Omron CX-Programmer project 新工程 (CX-Programmer 9.73)

# PLC 新PLC1: CPM2* 

## Global symbols (name address type ; comment)
0.00 BOOL  ; 系统工作/停止开
0.01 BOOL  ; 温度过高报警信号
0.03 BOOL  ; 湿度过高报警信号
0.05 BOOL  ; 烟雾报警信号
10.00 BOOL  ; 1
10.01 BOOL  ; 排风扇
10.02 BOOL  ; 烟雾报警信号
10.03 BOOL  ; 温度报警信号
10.04 BOOL  ; 系统运行灯
10.05 BOOL  ; 温度报警灯
10.06 BOOL  ; 湿度报警灯
10.07 BOOL  ; 烟雾报警灯
200.00 BOOL  ; 0点开信号
200.01 BOOL  ; 4点开信号
200.02 BOOL  ; 8点开信号
200.03 BOOL  ; 12点开信号
200.04 BOOL  ; 16点开信号
200.05 BOOL  ; 20点开信号
200.10 BOOL  ; 触发信号
232.00 BOOL  ; 系统运行

## Program 新程序1 (no task)
; 原创、欧姆龙PLC、CPM2A自身时钟六个时间段触发程序 / 简单程序，高手请飘过。 / 欧姆龙CPM2A六个时间段触发程序。 / 触发时间为0点，4点，8点，12点，16点，20点（可通过修改CMP20#的值修改触发时间）一分钟后断开。 / 触发次数也可通过增减CMP20来实现。 / 在实际应用中，当系统工作开关开启时，系统根据PLC时钟读取时间数据，在 0点、4点、8点、12点、16点、20点 置位对应的触发信号，并通过这些信号组合生成综合触发信号来驱动设备动作。当综合触发信号被置位时，系统进入运行状态并准备设备动作。系统确保在任一时刻，只有一个触发信号被置位，以保证动作独立执行。 / 系统还集成了安全监测功能，当温度过高信号、湿度过高信号或烟雾检测信号被触发时，温度报警灯、湿度报警灯或烟雾报警灯会点亮，同时通过温度报警输出或烟雾报警输出通知外部设备，以保护生产安全。若 0点触发信号被置位，启动设备初始动作；若 4点触发信号被置位，调整设备运行参数。此外，PLC时钟与实际时间保持同步，在 0点 准时置位 0点触发信号，准备设备运行。

### Section 段1

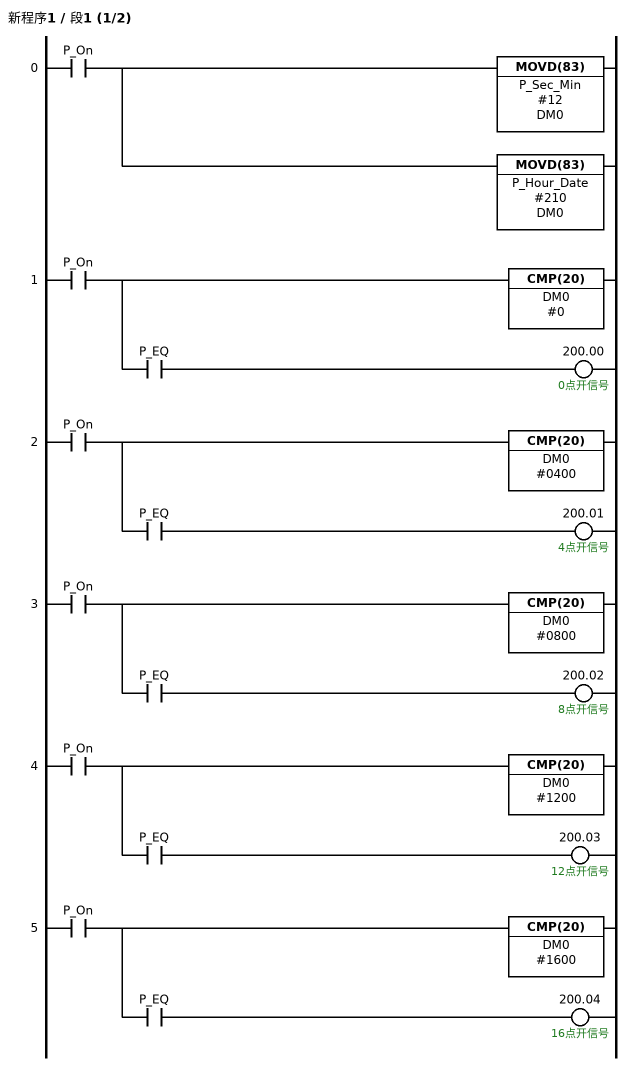
; rung 0
LD P_On
MOVD(83) P_Sec_Min #12 DM0
MOVD(83) P_Hour_Date #210 DM0
; rung 1
LD P_On
CMP(20) DM0 #0
AND P_EQ
OUT 200.00  ; 0点开信号
; rung 2
LD P_On
CMP(20) DM0 #0400
AND P_EQ
OUT 200.01  ; 4点开信号
; rung 3
LD P_On
CMP(20) DM0 #0800
AND P_EQ
OUT 200.02  ; 8点开信号
; rung 4
LD P_On
CMP(20) DM0 #1200
AND P_EQ
OUT 200.03  ; 12点开信号
; rung 5
LD P_On
CMP(20) DM0 #1600
AND P_EQ
OUT 200.04  ; 16点开信号

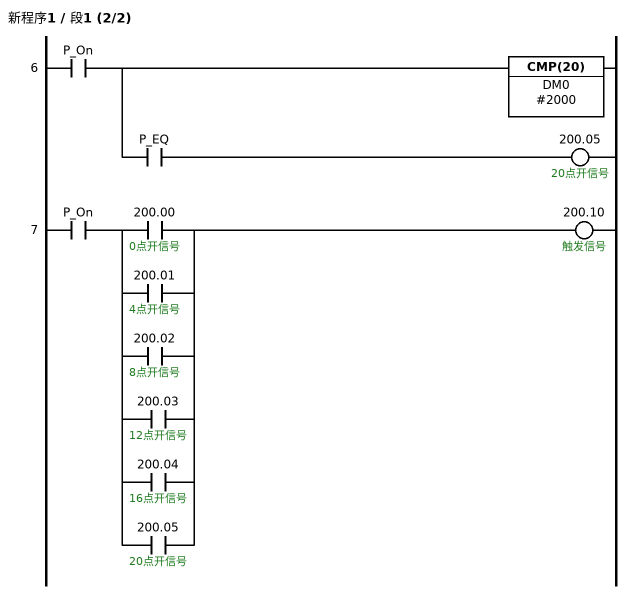
; rung 6
LD P_On
CMP(20) DM0 #2000
AND P_EQ
OUT 200.05  ; 20点开信号
; rung 7
LD P_On
LD 200.00  ; 0点开信号
OR 200.01  ; 4点开信号
OR 200.02  ; 8点开信号
OR 200.03  ; 12点开信号
OR 200.04  ; 16点开信号
OR 200.05  ; 20点开信号
ANDLD
OUT 200.10  ; 触发信号
; rung 8
END(01)